KUKA KRL program: Touchpoint_7_2.src

&ACCESS RVP
&REL 1
&PARAM TEMPLATE = C:\KRC\Roboter\Template\vorgabe
&PARAM EDITMASK = *
DEF Touchpoint_7_2 ( )


;FOLD INI
;FOLD BASISTECH INI
GLOBAL INTERRUPT DECL 3 WHEN $STOPMESS==TRUE DO IR_STOPM ( )
INTERRUPT ON 3
BAS (#INITMOV,0 )
;ENDFOLD (BASISTECH INI)
;ENDFOLD (INI)

;FOLD STARTPOSITION - BASE IS 0, TOOL IS 5, SPEED IS 15%, POSITION IS A1 5,A2 -90,A3 100,A4 5,A5 -10,A6 -5,E1 0,E2 0,E3 0,E4 0
$BWDSTART = FALSE
PDAT_ACT = {VEL 15,ACC 100,APO_DIST 50}
FDAT_ACT = {TOOL_NO 5,BASE_NO 0,IPO_FRAME #BASE}
BAS (#PTP_PARAMS,15)
PTP  {A1 5,A2 -90,A3 100,A4 5,A5 -10,A6 -5,E1 0,E2 0,E3 0,E4 0}
;ENDFOLD

;FOLD LIN SPEED IS 0.1 m/sec, INTERPOLATION SETTINGS IN FOLD
$VEL.CP=0.1
$ADVANCE=3
;ENDFOLD

BAS(#VEL_PTP,3)
PTP {X 342.707, Y 362.992, Z 432.358, A -116.805, B 80.034, C -131.472, E1 0, E2 0, E3 0, E4 0, S 'B010'}
BAS(#VEL_PTP,1)
PTP {X 342.707, Y 362.992, Z 402.358, A -116.805, B 80.034, C -131.472, E1 0, E2 0, E3 0, E4 0, S 'B010'}
BAS(#VEL_PTP,3)
PTP {X 342.707, Y 362.992, Z 432.358, A -116.805, B 80.034, C -131.472, E1 0, E2 0, E3 0, E4 0, S 'B010'}
PTP {A1 5, A2 -90, A3 100, A4 5, A5 -10, A6 -5, E1 0, E2 0, E3 0, E4 0} C_PTP

END
